FUNCTION_BLOCK ClearLinkEIP
VAR_INPUT
	bEnable : BOOL;
END_VAR
VAR_OUTPUT
	pulse AT %Q* : INT; //num pulses
	outputRegister AT %Q* : INT;
	brakeRelease AT %Q* : BOOL;
	
	A : BOOL; //direction (F = inwards, T = outwards)
	B : BOOL; //home bit
	clear : BOOL;
	
	contact AT %I* : BOOL;
	home AT %I* : BOOL;
	outerLimit AT %I* : BOOL;
	innerLimit AT %I* : BOOL;
	
	hlfb AT %I* : REAL;
	
	homeSet : BOOL;
	busy : BOOL;
	error : BOOL;
	
	position : LREAL;
	targetPos : LREAL;
END_VAR
VAR
	test : BOOL;
	pulseRequest : INT;
	
	pulser : TON;
	//pulseSeparator : TOF;
	
	minHoming : TON;
	resetTimer : TP;
	
	step : Homing; //(IDLE, HOME_UP, HOME_FINAL, DOWN, REDO_HOME, HOME_DONE);
	mode : (DISABLE, HOLD, TARGET, CONTINUOUS, RESET_ERR);
END_VAR
VAR_STAT CONSTANT
	resetTime : TIME := T#1000MS;
	pulseWidth : TIME := T#40MS;
	pulseSeparation : TIME := T#40MS;
	unitsPerPulse : INT := 800; //800 Teknic units per revolution
	distancePerPulse : INT := 5; //5mm per revolution
END_VAR

IF NOT bEnable THEN
	mode := DISABLE;
END_IF


outputRegister.0 := bEnable;
outputRegister.1 := A;
outputRegister.2 := B;
outputRegister.3 := clear;

resetTimer(IN:= , PT:= resetTime, Q=> clear, ET=> );
//pulseSeparator(IN:= busy, PT:= pulseSeparation, Q=> , ET=> );

//set the bool outputs, all are listed for readability
homeSet := homeSet;
busy := hlfb <> -9999;
error := error;

CASE mode OF
	DISABLE:
		//bEnable := FALSE;
		pulse := 0;
		pulseRequest := 0;
		
	HOLD:
		pulse := 0;
		pulseRequest := 0;
	
	TARGET:	
		test := WithinTolerance(position, targetPos, distancePerPulse);
		IF WithinTolerance(position, targetPos, distancePerPulse) THEN
			pulseRequest := 0;
			mode := HOLD;
			
		ELSIF NOT busy THEN
			//test := TRUE;
			A :=  position < targetPos;
			pulseRequest := TO_INT(ABS(position - targetPos)/distancePerPulse); //pulseAll();
			//pulseRequest := 1; //pulseSingle();
			
		END_IF
		
	CONTINUOUS:
		pulseRequest := 1;
		
	RESET_ERR:
		pulse := 0;
		pulseRequest := 0;
		resetTimer.IN := TRUE;
		
		IF resetTimer.Q THEN
			resetTimer.IN := FALSE;
			mode := HOLD;
		END_IF
		
END_CASE

IF home AND_THEN A THEN //block outwards motion
	position := 0;
	mode := HOLD;
	
ELSIF outerLimit AND_THEN A THEN //block outwards motion
	mode := HOLD;

ELSIF innerLimit AND_THEN NOT A THEN //block inwards motion
	mode := HOLD;
	
END_IF

sequence();

METHOD homingSequence : BOOL
minHoming(IN:= , PT:= T#1S, Q=> , ET=> );

IF NOT bEnable THEN
	mode := DISABLE;
	RETURN;
END_IF

CASE step OF
	Homing.IDLE:
		A := FALSE;
		B := FALSE;
		brakeRelease := TRUE;
		
		homeSet := FALSE;
		step := Homing.REDO;
		
	Homing.REDO: //let insertion drop to inner limit before homing
		A := FALSE;
		B := FALSE;
		brakeRelease := TRUE;
		
		IF NOT innerLimit THEN
			mode := CONTINUOUS;
			step := Homing.HOME_OUT;
		END_IF
	
	Homing.HOME_OUT:
		mode := CONTINUOUS;
	
		A := FALSE;
		B := TRUE;
		brakeRelease := TRUE;
		
		minHoming.IN := TRUE;
		
		IF NOT home AND minHoming.Q THEN
			minHoming.IN := FALSE;
			
			mode := HOLD;
			step := Homing.DONE;
		END_IF
		
	Homing.DONE:
		pulse := 0;
		A := FALSE;
		B := FALSE;
		brakeRelease := TRUE;
		
		position := 0;
		homeSet := TRUE;
		homingSequence := TRUE;
		
		mode := HOLD;
		step := Homing.IDLE;
	
END_CASE
END_METHOD

METHOD moveAbsolute : BOOL
VAR_INPUT
	newTarget : LREAL;
END_VAR
targetPos := newTarget;
mode := TARGET;
END_METHOD

METHOD moveContinuous : BOOL
VAR_INPUT
	direction : MC_Direction;
END_VAR
IF direction = MC_Negative_Direction THEN
	A := FALSE;
ELSIF direction = MC_Positive_Direction THEN
	A := TRUE;
END_IF

mode := CONTINUOUS;
END_METHOD

METHOD reset : BOOL
VAR_INPUT
END_VAR
mode := RESET_ERR;
END_METHOD

METHOD sequence : BOOL
VAR_INPUT
END_VAR
IF hlfb > -9999 THEN //is busy
	IF A THEN //positive
		position := position + (distancePerPulse * pulse);
	ELSE
		position := position - (distancePerPulse * pulse);
	END_IF
	pulse := 0;
	RETURN;
END_IF

//is free to accept new request
IF pulse = 0 (*AND NOT pulseSeparator.Q*) THEN
	pulse := pulseRequest;
	//pulseRequest := 0;
END_IF
END_METHOD

METHOD stop : BOOL
VAR_INPUT
END_VAR
mode := HOLD;
END_METHOD

END_FUNCTION_BLOCK

(* stored: Version 1.1.0.1, ProductVersion 3.1.4024.11
   POU ClearLinkEIP: Id {82d395c8-897a-4c3b-989f-b99dc8146760}, SpecialFunc None
   Folder Public Methods: Id {d29c5c5d-14f1-4972-8db5-81b3764b5246}
   Method homingSequence: Id {ed7f9015-f217-4688-b191-db86d43e2b15}
   Method moveAbsolute: Id {dc77def1-bef9-43df-afd0-8ca352bd4ae2}
   Method moveContinuous: Id {56e37924-ed1f-434c-b8b5-86f83bcd5e14}
   Method reset: Id {b78ab13d-678d-4b52-8830-ac5e90a85d68}
   Method sequence: Id {d3e76146-deb6-4a1c-bf00-057dae828590}
   Method stop: Id {b371037c-73c2-41cf-af60-cf703d5e079a} *)
